ABB RobotStudio station: Trabajo Robotica.rsstn

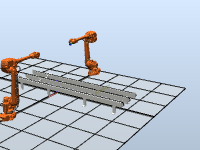
Station Trabajo Robotica (saved by RobotStudio 6.4.7152.140)
Controller IRB_4600_40kg_2.55m_2, task T_ROB1: task frame (RAPID world) sits at (2500, 0, 0) mm, rotated rx 0 ry 0 rz 180 deg in the station
Controller IRB_4600_40kg_2.55m_1, task T_ROB1: task frame (RAPID world) sits at (-2500, 0, 0) mm in the station
Controller IRB_4600_40kg_2.55m_1
  mechanical unit ROB_1: IRB4600_40_255__02, 6 joints, base frame (0, 0, 0) mm
Controller IRB_4600_40kg_2.55m_2
  mechanical unit ROB_1: IRB4600_40_255__02_2, 6 joints, base frame (0, 0, 0) mm
Layout (positions relative to the parent item):
  - IRB4600_40_255__02 [mechanism, from Robots\IRB4600_40_255__02.rslib] at (-2500, 0, 0) mm; joint values [0, 0, 0, 0, 0.5236, 0] (rad or m)
  - IRB4600_40_255__02_2 [mechanism, from Robots\IRB4600_40_255__02.rslib] at (2500, 0, 0) mm, rotated rx 0 ry 0 rz 180 deg; joint values [0, 0, 0, 0, 0.5236, 0] (rad or m)
  - 4800_3str_h2 [part, from Equipment\Conveyor 4800 3str h2.rslib] at (400, -1500, 0) mm, rotated rx 0 ry 0 rz 90 deg
  - AlimentadorCoches [smart component]
      signals: DI diNuevoCoche, DO doCochePosit
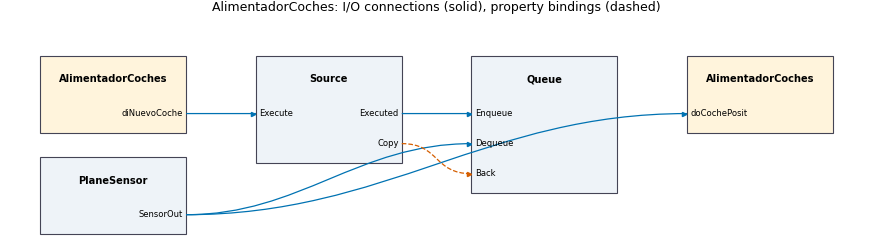
      connections:
        AlimentadorCoches.diNuevoCoche -> Source.Execute
        Source.Executed -> Queue.Enqueue
        PlaneSensor.SensorOut -> Queue.Dequeue
        PlaneSensor.SensorOut -> AlimentadorCoches.doCochePosit
        Source.Copy => Queue.Back
    - Source [smart component, from Components\Source.rslib]
        properties: Source=(none); Copy=(none); Parent=(none); Position=[0.8 0 0.3]; Orientation=[1.5707963267949 0 3.14159265358979]; Transient=false
    - Queue [smart component, from Components\Queue.rslib]
        properties: Back=(none); Front=(none); Queue={88de15b8-0fc9-49a3-9f74-bd66be803ec1};{707d295b-cad9-4ac1-bd48-2442d05ced9b};{40def8f1-bb45-40d3-af39-f83ca5696c45};{ef7d474d-35c4-4274-862a-19b279423ff9};{b5885754-f7c0-4be8-a7df-44c7500c3c4e};{d289849f-2ef8-4886-87b8-beb05382232c}; NumberOfObjects=1
    - PlaneSensor [smart component, from Components\PlaneSensor.rslib]
        properties: Origin=[0.45 2 0.48]; Axis1=[-1 0 0]; Axis2=[0 0 0.1]; SensedPart=(none)
      - _sensorPart_ [part]
    - LinearMover [smart component, from Components\LinearMover.rslib]
        properties: Object=Queue; Direction=[0 1 0]; Speed=1; Reference=Local; ReferenceObject=(none)
